// Implicitly generated code : DO NOT EDIT
FUNCTION CheckBounds : DINT
VAR_INPUT
    index, lower, upper : DINT;
END_VAR

// Implicitly generated code : Only an Implementation suggestion
{noflow}
IF index < lower THEN
    CheckBounds := lower;
ELSIF index > upper THEN
    CheckBounds := upper;
ELSE
    CheckBounds := index;
END_IF

{flow}

END_FUNCTION

(* stored: Version 1.1.0.1, ProductVersion 3.1.4024.12
   POU CheckBounds: Id {2b1b1979-3e46-01d5-3410-2262dec1abf1}, SpecialFunc CheckBounds *)
